(* CoDeSys 2.3.9.41 project: sample_plc160m.pro *)
(* Libraries: SysLibMem.lib 20.2.06 13:31:12, SysLibCom.lib 20.2.06 13:31:08, Owen\PID_Regulators.lib 28.12.06 17:47:54, Util.lib 18.5.10 15:14:28, STANDARD.LIB 4.10.05 11:14:46, SysLibSockets.lib 20.2.06 13:31:14 *)

(* PLC configuration (modules and I/O channels)
Fast discrete inputs [I_SIMPLE_INPUT] node 0, in %IB0 out %QB0 {Filtrationtime = 10}
  AT %IX0.0 [BitInput] Discrete input 1
  AT %IX0.1 [BitInput] Discrete input 2
  AT %IX0.2 [BitInput] Discrete input 3
  AT %IX0.3 [BitInput] Discrete input 4
Discrete inputs [ID130] node 1, in %IB1 out %QB1 {Filtrationtime_GeneralINP = 10; Visibility = No; PinCount = 12}
  AT %IB1.0 [ByteInput] 8 discrete inputs
  AT %IB1.1 [ByteInput] 4 discrete inputs
Discrete outputs [ID131] node 2, in %IB2 out %QB2 {SafeValueByte = 0; SafeValueByteM = 0; Visibility = No; PinCount = 12}
  AT %QB2.0 [ByteOutput] 8 discrete outputs
  AT %QB2.1 [ByteOutput] 4 discrete outputs
Fast analog inputs [ID125] node 3, in %IB3 out %QB3 {Flt_Comm = 50Hz 2Por}
  AT %IR3.0 [FloatInputP] AI #1 {AIN_TYPE = 4-20 mA; Peak_Filtr = 200; Flt_Ch = Off; TauRC = 10; MinFV = 0; MaxFV = 131}
  AT %IR3.1 [FloatInputP] AI #2 {AIN_TYPE = 4-20 mA; Peak_Filtr = 200; Flt_Ch = Off; TauRC = 10; MinFV = 0; MaxFV = 20000.0}
  AT %IR3.2 [FloatInputP] AI #3 {AIN_TYPE = 4-20 mA; Peak_Filtr = 200; Flt_Ch = Off; TauRC = 10; MinFV = 0; MaxFV = 20000.0}
  AT %IR3.3 [FloatInputP] AI #4 {AIN_TYPE = 4-20 mA; Peak_Filtr = 200; Flt_Ch = Off; TauRC = 10; MinFV = 0; MaxFV = 20000.0}
  AT %IR3.4 [FloatInputP] AI #5 {AIN_TYPE = 4-20 mA; Peak_Filtr = 200; Flt_Ch = Off; TauRC = 10; MinFV = 0; MaxFV = 20000.0}
  AT %IR3.5 [FloatInputP] AI #6 {AIN_TYPE = 0-10V; Peak_Filtr = 200; Flt_Ch = Off; TauRC = 10; MinFV = 0; MaxFV = 10}
  AT %IR3.6 [FloatInputP] AI #7 {AIN_TYPE = 4-20 mA; Peak_Filtr = 200; Flt_Ch = Off; TauRC = 10; MinFV = 0; MaxFV = 20000.0}
  AT %IR3.7 [FloatInputP] AI #8 {AIN_TYPE = 4-20 mA; Peak_Filtr = 200; Flt_Ch = Off; TauRC = 1000; MinFV = 0; MaxFV = 130}
  AT %IW3.8 [WordInput] AI read time (10ms)
Analog outputs [ID126] node 4, in %IB4 out %QB4
  AT %QR4.0 [FloatOutputP] AO #1 {AOUT_TYPE = 4-20 mA; SafeValueREAL = 0.0}
  AT %QR4.1 [FloatOutputP] AO #2 {AOUT_TYPE = 0-10V; SafeValueREAL = 0.0}
  AT %QR4.2 [FloatOutputP] AO #3 {AOUT_TYPE = 4-20 mA; SafeValueREAL = 0.0}
  AT %QR4.3 [FloatOutputP] AO #4 {AOUT_TYPE = 0-10V; SafeValueREAL = 0.0}
Special input [ID103] node 5, in %IB5 out %QB5 {Filtrationtime = 1000; PinCount = 1; WatchDogPeriod = 400; PollPeriod = 3000; Visibility = No}
  AT %IX5.0 [BitInput] Special input
Special output [ID104] node 6, in %IB6 out %QB6 {Visibility = No; PinCount = 1}
  AT %QX6.0 [BitOutput] Special output
Modbus [MODBUS_ID302] node 0, in %IB7.0 out %QB7.0
  TCP [TCP_ID221] node 0, in %IB7.0.0 out %QB7.0.0 {RemotePort = 502; Visibility = No}
2 byte [Register] node 1, in %IB7.1 out %QB7.1
  hmi_cmd AT %QW7.1.0 [WordOutput]
2 byte [Register] node 2, in %IB7.2 out %QB7.2
  hmi_arg0 AT %QW7.2.0 [WordOutput]
2 byte [Register] node 3, in %IB7.3 out %QB7.3
  hmi_arg1 AT %QW7.3.0 [WordOutput]
Float [Float] node 4, in %IB7.4 out %QB7.4
  hmi_tension AT %QD7.4.0 [FloatOutput]
Float [Float] node 5, in %IB7.5 out %QB7.5
  hmi_pos AT %QD7.5.0 [FloatOutput]
Float [Float] node 6, in %IB7.6 out %QB7.6
  hmi_pos_setpoint AT %QD7.6.0 [FloatOutput]
Float [Float] node 7, in %IB7.7 out %QB7.7
  hmi_speed_lim AT %QD7.7.0 [FloatOutput]
8 bits [8Bit] node 8, in %IB7.8 out %QB7.8
  AT %QB7.8.0 [ByteOutput]
8 bits [8Bit] node 9, in %IB7.9 out %QB7.9
  AT %QB7.9.0 [ByteOutput]
2 byte [Register] node 10, in %IB7.10 out %QB7.10
  hmi_loop_state AT %QW7.10.0 [WordOutput]
Float [Float] node 11, in %IB7.11 out %QB7.11
  hmi_measured_speed AT %QD7.11.0 [FloatOutput]
sim_bus_addr AT %QD8.0 [DWordOutput] Last address
sim_bus_code AT %QW8.1 [WordOutput] Last error
RS-232 [COM2_USART] node 0, in %IB8.0 out %QB8.0 {CommunicationSpeed = 11520; Parity = NO PARITY CHECK; BitLength = 8 bits; StopLength = One stop bit; InterfaceType = RS232; FrameOriented = RTU; Timeout = 0; Visibility = No}
Universal Modbus device [ID2000] node 1, in %IB8.1 out %QB8.1 {ModuleIP = 10:0:0:223; ServiceTimeout = 150; TCPport = 502; NetMode = Serial; ModuleSlaveAddress = 1; RequestType = By poll time; PeriodOfService = 10; Visibility = No; RepeatCounter = 0; ByteSequence = Native}
  AT %QB8.1.0 [ComChannel] Command (0xff - Start)
  Real input module [ID2007] node 0, in %IB8.1.0 out %QB8.1.0 {ModbusAddress = 0; Command_read_regs = Read holding Registers  (0x03); Visibility = No}
    sim_force AT %ID8.1.0.0 [FloatInput]
  Real input module [ID2007] node 1, in %IB8.1.1 out %QB8.1.1 {ModbusAddress = 2; Command_read_regs = Read holding Registers  (0x03); Visibility = No}
    sim_pos AT %ID8.1.1.0 [FloatInput]
  Real output module [ID2008] node 2, in %IB8.1.2 out %QB8.1.2 {ModbusAddress = 0; Command_write_regs = Preset multiple Registers (0x10); Visibility = No}
    sim_speed AT %QD8.1.2.0 [FloatOutput]
AT %IW9.0 [WordInput] Cycle time in 100 mks
AT %IW9.1 [WordInput] Time to backup power down, s
AT %ID9.2 [FloatInput] Temp inside PLC
AT %IX9.3 [BitInput] Power status
AT %IX9.4 [BitInput] CPU is overloaded, optimize your programm or increase PLC cycle
AT %IW9.5 [WordInput] Free processor resourse mks in 1 cycle
*)

(* Global variable list: Global_Variables *)
VAR_GLOBAL
	_SIMMODE: BOOL;
END_VAR

(* Data type *)
TYPE EWM_CTRL_MODE : (
	IDLE, LOOP, MANUAL_THROTTLING, SET
);
END_TYPE

(* Data type *)
TYPE PLC_CMD : (NOP, SET_POSITIONS, SET_THROTTLE, SET_EBYPASS, SET_MODE, GOTO_POS, START_LOOP, SET_SPEED);
END_TYPE

(* Data type *)
TYPE RANGE :
STRUCT
	start, end: REAL;
END_STRUCT
END_TYPE

(* Data type *)
TYPE SIM_DATA_CLUMP :
STRUCT
	LDT: REAL;
	SPEED: REAL;
	TENSION: REAL;
	EWM_ENABLE, EWM_START: BOOL;
	EWM_POS, EWM_SPEED: REAL;
END_STRUCT
END_TYPE

(* Data type in Tilkom *)
TYPE TLK_CMD : (
	READ_VERSION := 66, GET_CURRENT_TIME, SET_CURRENT_TIME, GET_MESSAGE,

	START_MEASURING := 101, STOP_MEASURING, GET_ID, READ_BASE,
	READ_SPEED, READ_TEMP, READ_COMPLEX, STREAM_BASE, SET_PARAM
);
END_TYPE

(* Data type in Tilkom *)
TYPE TLK_XSTATE : (
	TLKX_IDLE,
	TLKX_START_QRY,
	TLKX_START_ACK,
	TLKX_VALUE_QRY,
	TLKX_VALUE_RSP,
	TLKX_SUCCESS,
	TLKX_STOP_QRY,
	TLKX_STOP_ACK,
	TLKX_ERROR
);
END_TYPE

(* POU PLC_PRG, ST *)
PROGRAM PLC_PRG
;
END_PROGRAM

(* Visualisation Vis
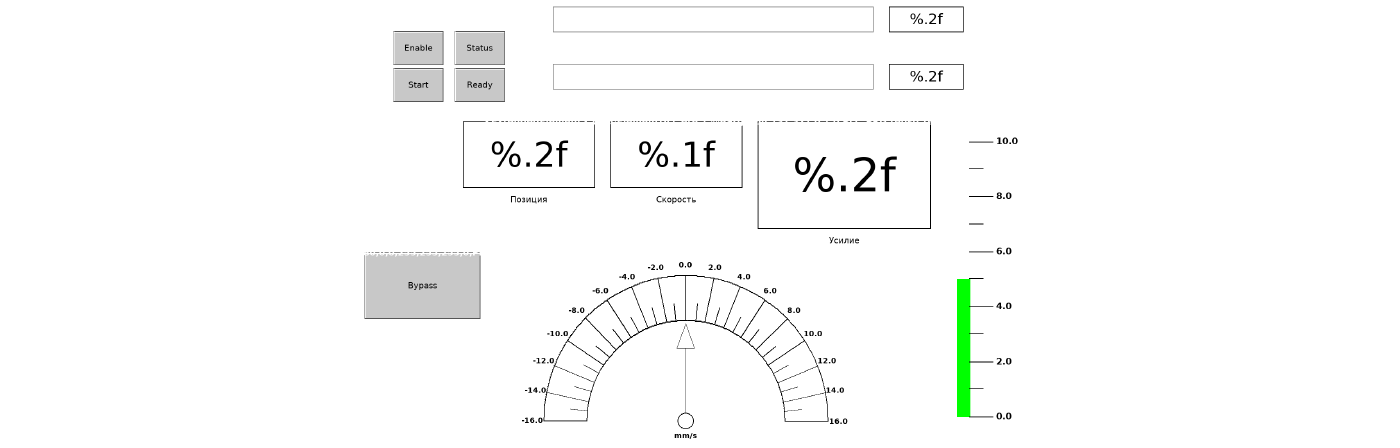
button at (45,50)-(106,91): text "Enable"; toggles EWM_ENABLE
button at (120,95)-(181,136): text "Ready"; toggles EWM_READY
button at (45,95)-(106,136): text "Start"; toggles EWM_START
button at (120,50)-(181,91): text "Status"; toggles EWM_STATUS
rectangle at (130,160)-(291,241): text "%.2f"; shows LDT_POS
rectangle at (310,160)-(471,241): text "%.1f"; shows PLC_PRG.speed_mtr.SPEED
rectangle at (490,160)-(701,291): text "%.2f"; shows PLC_PRG.tenso_reader.value
rectangle at (130,240)-(291,271): text "Позиция"
rectangle at (310,240)-(471,271): text "Скорость"
rectangle at (490,290)-(701,321): text "Усилие"
button at (10,320)-(151,401): text "Bypass"; toggles EBYPASS_VALVE
rectangle at (650,20)-(741,51): text "%.2f"; shows PLC_PRG.speed_out.IN
rectangle at (650,90)-(741,121): text "%.2f"; shows PLC_PRG.pos_out.IN
group at (200,320)-(601,551)
  rectangle at (0,0)-(1,1): text "{ExtendedElement},Visu\ElementDLL.ete,0,@Zeigerinstrument,401,180,0,0,255,255,255,0,PLC_PRG.speed_mtr.SPEED,mm/s,%.1f,0,1,1,1,2,-16,16,0,0,0,0,0,0,0,-11,80,700,Arial,1,0,0,255,255,255,,0,0,0,0,"
  rectangle at (0,193)-(29,207): text "-16.0"
  rectangle at (4,157)-(33,171): text "-14.0"
  rectangle at (14,122)-(43,136): text "-12.0"
  rectangle at (31,90)-(60,104): text "-10.0"
  rectangle at (57,62)-(80,76): text "-8.0"
  rectangle at (86,39)-(109,53): text "-6.0"
  rectangle at (118,22)-(141,36): text "-4.0"
  rectangle at (153,11)-(176,25): text "-2.0"
  rectangle at (191,8)-(210,22): text "0.0"
  rectangle at (227,11)-(246,25): text "2.0"
  rectangle at (262,22)-(281,36): text "4.0"
  rectangle at (294,39)-(313,53): text "6.0"
  rectangle at (323,62)-(342,76): text "8.0"
  rectangle at (343,90)-(368,104): text "10.0"
  rectangle at (360,122)-(385,136): text "12.0"
  rectangle at (370,157)-(395,171): text "14.0"
  rectangle at (374,194)-(399,208): text "16.0"
  rectangle at (185,211)-(217,225): text "mm/s"
  polygon at (190,85)-(211,201): angle ((PLC_PRG.speed_mtr.SPEED * 1.0)-0) * 5.625
group at (710,160)-(841,531)
  rectangle at (0,0)-(1,1): text "{ExtendedElement},Visu\ElementDLL.ete,1,@Bargraph,131,371,0,1,0,PLC_PRG.tenso_reader.value,,%.1f,1,2,0,10,0,0,0,0,0,0,0,-13,16,700,Arial,0,255,0,255,0,0,0,0,0,0,0,0,0,,0,0,0,"
  rectangle at (21,185)-(36,346): alarm colour if (PLC_PRG.tenso_reader.value) < 0; top ((PLC_PRG.tenso_reader.value * 1.0) - 5)  * -32.2
  rectangle at (64,335)-(122,356): text "0.0"
  rectangle at (64,271)-(122,292): text "2.0"
  rectangle at (64,206)-(122,227): text "4.0"
  rectangle at (64,142)-(122,163): text "6.0"
  rectangle at (64,77)-(122,98): text "8.0"
  rectangle at (64,13)-(122,34): text "10.0"
49 more shapes without text or variables
*)
